FUNCTION_BLOCK Mc3Axis_TcEvents EXTENDS CyclicComponent IMPLEMENTS I_EventReactionTcEvents
VAR
	Axis   : I_Mc3Axis;
	Events : TcEventClass(CONCAT(Name, ' Events'));
END_VAR

METHOD CyclicLogic
IF Axis.MotionTasks.Error THEN
	Events.Arguments(E_McAxis.AxisError).Clear().AddString(Axis.MotionTasks.ErrorTask).AddString(TO_STRING(Axis.MotionTasks.ErrorId));
	Events.RaiseEvent(E_McAxis.AxisError);
END_IF
END_METHOD

(*FB_Init is always available implicitly and it is used primarily for initialization.
The return value is not evaluated. For a specific influence, you can also declare the
methods explicitly and provide additional code there with the standard initialization
code. You can evaluate the return value.*)
METHOD FB_Init : BOOL
VAR_INPUT
	(* TRUE: the retain variables are initialized (reset warm / reset cold)*)
	bInitRetains : BOOL;

	(* TRUE: the instance will be copied to the copy code afterward (online change)   *)
	bInCopyCode : BOOL;
	Name		: T_MaxString;
	Axis		: I_Mc3Axis;
END_VAR
THIS^.Axis := Axis;
Events.GenerateTcEvents(Axis.Name, ADR(TC_events.MCAxis), SIZEOF(ST_MCAxis));
END_METHOD

METHOD GetHighestActiveEventReaction : DINT
GetHighestActiveEventReaction := Events.GetHighestActiveEventReaction();
END_METHOD

METHOD GetHighestActiveEventSeverity : TcEventSeverity
GetHighestActiveEventSeverity := Events.GetHighestActiveEventSeverity();
END_METHOD

METHOD Reset
Events.Reset();
END_METHOD

METHOD SetEventReactions
VAR_INPUT
	Verbose	 : DINT := 0;
	Info	 : DINT := 1;
	Warning	 : DINT := 2;
	Error	 : DINT := 3;
	Critical : DINT := 4;
END_VAR
Events.SetEventReactions(Verbose,
						 Info,
						 Warning,
						 Error,
						 Critical);
END_METHOD

END_FUNCTION_BLOCK

(* stored: Version 1.1.0.1, ProductVersion 3.1.4026.20
   POU Mc3Axis_TcEvents: Id {300f83e3-dc12-4b14-834a-357620f90932}, SpecialFunc None
   Folder Events: Id {0e71a3cb-493a-4a64-9c1b-96f7fc41275f}
   Method CyclicLogic: Id {77ed7bff-bf83-41c9-bf40-4783290eafad}
   Method FB_Init: Id {f5a173e1-1d13-40e3-ad55-9c5be5f11900}
   Method GetHighestActiveEventReaction: Id {2db2ee6a-d6b6-4a4d-8632-d6a3531323aa}
   Method GetHighestActiveEventSeverity: Id {29b60752-7cf3-4aa3-8a60-1bc8dd5c89d2}
   Method Reset: Id {85c35942-06e5-4635-ac7f-4cd4b13041f3}
   Method SetEventReactions: Id {0989abbb-1f41-4c23-9df8-88d018483976} *)
